FUNCTION_BLOCK ConvertFunctions EXTENDS TcUnit.FB_TestSuite
VAR
END_VAR

AnyTypeToStringFunction();
StringToAnyFunction();

METHOD AnyTypeToStringFunction : BOOL
VAR
	stringVar : T_MaxString := 'test';
	intVar : INT := 42;
	realVar : REAL := 3.14;
END_VAR
TcUnit.TEST('ANY to STRING');

AssertEquals_STRING(
	Expected := 'test',
	Actual := AnyToString(stringVar),
	Message := 'Should convert STRING var to STRING');

AssertEquals_STRING(
	Expected := '42',
	Actual := AnyToString(intVar),
	Message := 'Should convert INT var to STRING');

AssertEquals_STRING(
	Expected := '3.14',
	Actual := AnyToString(realVar),
	Message := 'Should convert REAL var to STRING');
	
TEST_FINISHED();
END_METHOD

METHOD StringToAnyFunction : BOOL
VAR
	stringVar : T_MaxString;
	intVar : INT;
	realVar : REAL;
END_VAR
TcUnit.TEST('STRING to ANY');

StringToAny('this is test', stringVar);
StringToAny('42', intVar);
StringToAny('3.14', realVar);

AssertEquals_STRING(
	Expected := 'this is test',
	Actual := stringVar,
	Message := 'Should return correct STRING value');

AssertEquals_INT(
	Expected := 42,
	Actual := intVar,
	Message := 'Should return correct INT value');

AssertEquals_REAL(
	Expected := 3.14,
	Actual := realVar,
	Delta := 0.001,
	Message := 'Should return correct REAL value');

TEST_FINISHED();
END_METHOD

END_FUNCTION_BLOCK

(* stored: Version 1.1.0.1, ProductVersion 3.1.4024.12
   POU ConvertFunctions: Id {5c60e2d6-28aa-0817-3ab9-bc38d45e25ab}, SpecialFunc None
   Method AnyTypeToStringFunction: Id {88310384-b69f-02db-2220-3da8999f0eeb}
   Method StringToAnyFunction: Id {a36c0b1c-36fd-0119-07a2-92b4f80d3142} *)
